// TIA Portal V16 export
// export: Created 2023-03-29T11:03:21.4749485Z, ExportSetting WithDefaults, DisplayName Totally Integrated Automation Portal, DisplayVersion V16 Update 6, DisplayName TIA Portal Version Control Interface, DisplayVersion V16 Update 2, DisplayName TIA Portal Openness, DisplayVersion V16 Update 6, DisplayName STEP 7 Professional, DisplayVersion V16 Update 6, DisplayName STEP 7 Safety, DisplayVersion V16, DisplayName WinCC Advanced, DisplayVersion V16 Update 6
FUNCTION "Start_upPower" : Void   // FC22, LAD
TITLE = Start po restarcie
{ S7_Optimized_Access := 'TRUE' }
AUTHOR : rtecmer
VERSION : 0.1
// opóznienie aktualizacji stanów gotowości itp.
// stored: AutoNumber true, IsIECCheckEnabled false, SetENOAutomatically false, UDAEnableTagReadback false
   VAR_INPUT
      KT1 : Time;   // Czas timera
   END_VAR
   VAR_IN_OUT
      TMR1 : TON_TIME;
      isPowerOK : Bool;
   END_VAR
BEGIN

REGION Network 1
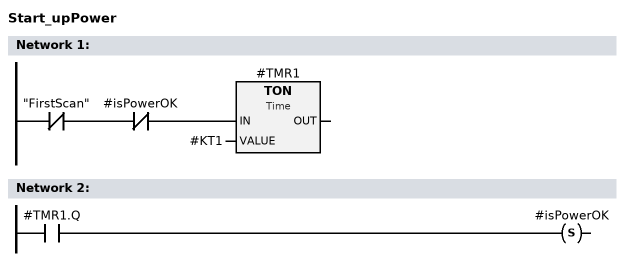
   #TMR1(IN := NOT "FirstScan" AND NOT #isPowerOK, PT := #KT1);   // TON coil
END_REGION

REGION Network 2
   RUNG wire#powerrail
      Contact( #TMR1.Q )
      S_Coil( #isPowerOK )
   END_RUNG
   // the same network as SCL:
   IF #TMR1.Q THEN #isPowerOK := TRUE; END_IF;
END_REGION
END_FUNCTION
